KUKA KRL data list: rReal.dat

&ACCESS RV1
&PARAM DISKPATH = Program/KukaMiling/Dat
DEFDAT  rReal PUBLIC


DECL GLOBAL INT grToolHolderDist=90

ENDDAT
